FUNCTION_BLOCK CNV_MDL_ASS (* Simple Conveyor Model for 1 Workpiece *)
  (* Standard: 61499-1; Classification: Simulation *)
  (* Version 1.0, 2018-05-09, JHC, Holobloc Inc, Added ECC, EMPTY; simplified algorithms for documentation. *)
  (* Version 0.0, 2004-09-20, JHC, Rockwell Automation, Simplified from CNV_MDL. *)
  PACKAGE fb.rt.Conveyer;
  IMPORT fb.datatype.*;
  IMPORT fb.rt.*;
  IMPORT fb.rt.mva.VSTYLE;
  (* Compiler Java Sun JDK 1.7.0 *)
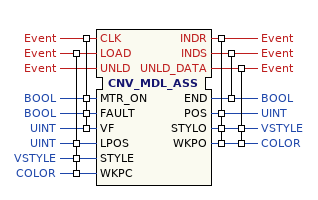
  EVENT_INPUT
    CLK WITH MTR_ON, VF, FAULT; (* Simulation Clock Event *)
    LOAD WITH STYLE, WKPC, LPOS; (* Load Workpiece if at HOME position *)
    UNLD; (* Unload Workpiece if at END position *)
  END_EVENT
  EVENT_OUTPUT
    INDR WITH POS, STYLO, WKPO; (* Change in Rendering Data *)
    INDS WITH END; (* Change in Sensor Data *)
    UNLD_DATA WITH STYLO, WKPO;
  END_EVENT
  VAR_INPUT
    MTR_ON : BOOL; (* Motor ON command *)
    FAULT : BOOL; (* Fault Condition *)
    VF : UINT; (* Conveyor Speed in % per CLK event *)
    LPOS : UINT; (* Load Position in % of Conveyor Length *)
    STYLE : VSTYLE := NONE; (* Input Workpiece style *)
    WKPC : COLOR := yellow; (* Input Workpiece Color *)
  END_VAR
  VAR_OUTPUT
    END : BOOL; (* Workpiece at End Position *)
    POS : UINT; (* Workpiece Position in % of Conveyor Length *)
    STYLO : VSTYLE := NONE; (* Currently loaded workpiece style *)
    WKPO : COLOR := blue; (* Currently loaded workpiece color *)
  END_VAR
  VAR
    EMPTY : BOOL := TRUE; (* STYLO = VSTYLE#NONE *)
  END_VAR
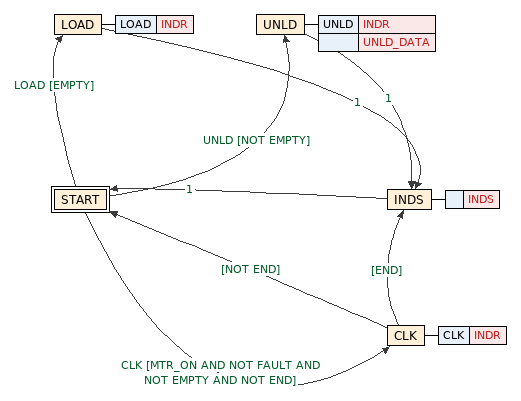
  EC_STATES
    START;
    LOAD : LOAD -> INDR;
    UNLD : UNLD -> INDR, -> UNLD_DATA;
    CLK : CLK -> INDR;
    INDS : -> INDS; (* Sensor change indication *)
  END_STATES
  EC_TRANSITIONS
    START TO CLK := CLK [MTR_ON AND NOT FAULT AND NOT EMPTY AND NOT END];
    START TO LOAD := LOAD [EMPTY];
    START TO UNLD := UNLD [NOT EMPTY];
    INDS TO START := 1;
    LOAD TO INDS := 1;
    UNLD TO INDS := 1;
    CLK TO INDS := [END];
    CLK TO START := [NOT END];
  END_TRANSITIONS
  ALGORITHM LOAD IN Java:
POS.value = Math.min(100,LPOS.value);
END.value = (POS.value==100)&&(STYLE.value != VSTYLE.NONE);
STYLO.value = STYLE.value;
WKPO.value = WKPC.value;
EMPTY.value = (STYLE.value == VSTYLE.NONE);
  END_ALGORITHM
  ALGORITHM UNLD IN Java:
STYLO.value=VSTYLE.NONE;
END.value = false;
EMPTY.value = true;
  END_ALGORITHM
  ALGORITHM CLK IN Java:
POS.value += VF.value;
if(POS.value>=100){
POS.value=100;
END.value=true;}
  END_ALGORITHM
END_FUNCTION_BLOCK
